// TIA Portal V18 export
// export: Created 2026-06-07T00:00:00Z, ExportSetting WithDefaults
VAR_GLOBAL   // PLC tag table "AI_Tags"
   Clock_1Hz AT %M0.5 : Bool;   // Clock_1Hz Modbus Tag
   FirstScan AT %M1.0 : Bool;   // FirstScan Modbus Tag
   MB_Write_Req AT %M10.0 : Bool;   // MB_Write_Req Modbus Tag
   MB_Read_Req AT %M10.1 : Bool;   // MB_Read_Req Modbus Tag
   MB_Write_Done AT %M10.2 : Bool;   // MB_Write_Done Modbus Tag
   MB_Write_Busy AT %M10.3 : Bool;   // MB_Write_Busy Modbus Tag
   MB_Write_Error AT %M10.4 : Bool;   // MB_Write_Error Modbus Tag
   MB_Read_Done AT %M10.5 : Bool;   // MB_Read_Done Modbus Tag
   MB_Read_Busy AT %M10.6 : Bool;   // MB_Read_Busy Modbus Tag
   MB_Read_Error AT %M10.7 : Bool;   // MB_Read_Error Modbus Tag
   MB_Write_Status AT %MW12 : Word;   // MB_Write_Status Modbus Tag
   MB_Read_Status AT %MW14 : Word;   // MB_Read_Status Modbus Tag
END_VAR
